// TIA Portal project "TEST_VENDRAME_ALESSANDRO" (V15)

(* hardware
DEVICE "S7-1200 station_1"  S7-1200 Station
   slot 0: "Rack_0"  S7-1200 Rack  Rack  V1.0
   slot 1: "PLC_1"  CPU 1215C DC/DC/DC  6ES7 215-1AG40-0XB0  V4.2
DEVICE "HMI_2"  KTP700 Basic PN
   slot 0: "HMI_2"  KTP700 Basic PN  6AV2 123-2GB03-0AX0  15.0.0.0
   slot 1: "HMI_RT_2"  KTP700 Basic PN  6AV2 123-2GB03-0AX0  15.0.0.0
   slot 5: "HMI_2.IE_CP_1"  PROFINET Interface  15.0.0.0
      slot 1: "PROFINET Interface_1"  PROFINET Interface
         slot 1: "Port_1"  Port
*)

// ===== PLC "PLC_1"  CPU 1215C DC/DC/DC =====

VAR_GLOBAL   // PLC tag table "Default tag table"
   "Clock_Byte" AT %MB666 : Byte;
   "1Hz_Clock" AT %M666.5 : Bool;
   "Clock_5Hz" AT %M666.1 : Bool;
   "Clock_2.5Hz" AT %M666.2 : Bool;
   "Clock_2Hz" AT %M666.3 : Bool;
   "Clock_1.25Hz" AT %M666.4 : Bool;
   "Clock_1Hz" AT %M666.5 : Bool;
   "Clock_0.625Hz" AT %M666.6 : Bool;
   "Clock_0.5Hz" AT %M666.7 : Bool;
END_VAR

DATA_BLOCK "GARA"   // DB1
{ S7_Optimized_Access := 'TRUE' }
VERSION : 0.1
   VAR
      TIMER_START : Bool;
      TIMER_STOP : Bool;
      TIMER_RESET : Bool;
      TIMER_TIME : Real;
      TEMPO_ATLETA_1 : Real;
      TEMPO_ATLETA_2 : Real;
      TEMPO_ATLETA_3 : Real;
      TEMPO_ATLETA_4 : Real;
      TEMPO_ATLETA_5 : Real;
      TEMPO_ATLETA_6 : Real;
      TEMPO_ATLETA_7 : Real;
      TEMPO_ATLETA_8 : Real;
      TimerStop_Atleta_1 : Bool;
      TimerStop_Atleta_2 : Bool;
      TimerStop_Atleta_3 : Bool;
      TimerStop_Atleta_4 : Bool;
      TimerStop_Atleta_5 : Bool;
      TimerStop_Atleta_6 : Bool;
      TimerStop_Atleta_7 : Bool;
      TimerStop_Atleta_8 : Bool;
      Race_Time : Real;
   END_VAR
BEGIN
END_DATA_BLOCK

ORGANIZATION_BLOCK "Main"   // OB1, LAD, ProgramCycle
TITLE = "Main Program Sweep (Cycle)"
{ S7_Optimized_Access := 'TRUE' }
VERSION : 0.1
   VAR_INPUT
      Initial_Call : Bool;   // Initial call of this OB
      Remanence : Bool;   // =True, if remanent data are available
   END_VAR
BEGIN

REGION Network 1
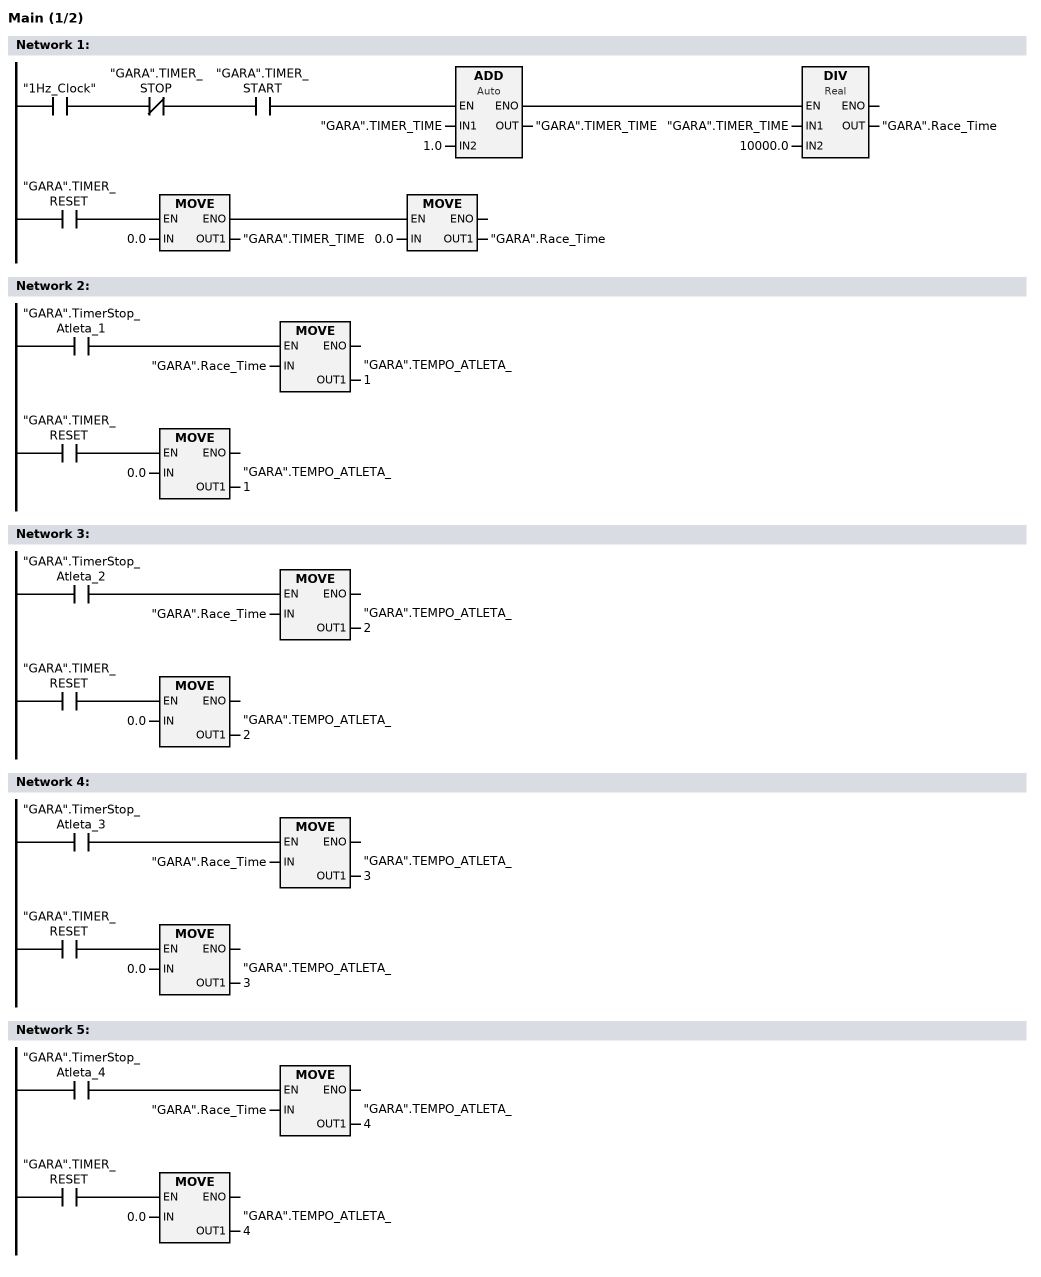
   RUNG wire#powerrail
      Contact( "1Hz_Clock" )
      I_Contact( "GARA".TIMER_STOP )
      Contact( "GARA".TIMER_START )
      Add(in1 := "GARA".TIMER_TIME, in2 := 1.0, out => "GARA".TIMER_TIME)
      { S7_Templates := "SrcType := Real" } Div(in1 := "GARA".TIMER_TIME, in2 := 10000.0, out => "GARA".Race_Time)
   END_RUNG
   RUNG wire#powerrail
      Contact( "GARA".TIMER_RESET )
      Move(in := 0.0, out1 => "GARA".TIMER_TIME)
      Move(in := 0.0, out1 => "GARA".Race_Time)
   END_RUNG
   // the same network as SCL:
   IF "1Hz_Clock" AND NOT "GARA".TIMER_STOP AND "GARA".TIMER_START THEN
       "GARA".TIMER_TIME := "GARA".TIMER_TIME + 1.0;
       "GARA".Race_Time := "GARA".TIMER_TIME / 10000.0;
   END_IF;
   IF "GARA".TIMER_RESET THEN
       "GARA".TIMER_TIME := 0.0;
       "GARA".Race_Time := 0.0;
   END_IF;
END_REGION

REGION Network 2
   RUNG wire#powerrail
      Contact( "GARA".TimerStop_Atleta_1 )
      Move(in := "GARA".Race_Time, out1 => "GARA".TEMPO_ATLETA_1)
   END_RUNG
   RUNG wire#powerrail
      Contact( "GARA".TIMER_RESET )
      Move(in := 0.0, out1 => "GARA".TEMPO_ATLETA_1)
   END_RUNG
   // the same network as SCL:
   IF "GARA".TimerStop_Atleta_1 THEN "GARA".TEMPO_ATLETA_1 := "GARA".Race_Time; END_IF;
   IF "GARA".TIMER_RESET THEN "GARA".TEMPO_ATLETA_1 := 0.0; END_IF;
END_REGION

REGION Network 3
   RUNG wire#powerrail
      Contact( "GARA".TimerStop_Atleta_2 )
      Move(in := "GARA".Race_Time, out1 => "GARA".TEMPO_ATLETA_2)
   END_RUNG
   RUNG wire#powerrail
      Contact( "GARA".TIMER_RESET )
      Move(in := 0.0, out1 => "GARA".TEMPO_ATLETA_2)
   END_RUNG
   // the same network as SCL:
   IF "GARA".TimerStop_Atleta_2 THEN "GARA".TEMPO_ATLETA_2 := "GARA".Race_Time; END_IF;
   IF "GARA".TIMER_RESET THEN "GARA".TEMPO_ATLETA_2 := 0.0; END_IF;
END_REGION

REGION Network 4
   RUNG wire#powerrail
      Contact( "GARA".TimerStop_Atleta_3 )
      Move(in := "GARA".Race_Time, out1 => "GARA".TEMPO_ATLETA_3)
   END_RUNG
   RUNG wire#powerrail
      Contact( "GARA".TIMER_RESET )
      Move(in := 0.0, out1 => "GARA".TEMPO_ATLETA_3)
   END_RUNG
   // the same network as SCL:
   IF "GARA".TimerStop_Atleta_3 THEN "GARA".TEMPO_ATLETA_3 := "GARA".Race_Time; END_IF;
   IF "GARA".TIMER_RESET THEN "GARA".TEMPO_ATLETA_3 := 0.0; END_IF;
END_REGION

REGION Network 5
   RUNG wire#powerrail
      Contact( "GARA".TimerStop_Atleta_4 )
      Move(in := "GARA".Race_Time, out1 => "GARA".TEMPO_ATLETA_4)
   END_RUNG
   RUNG wire#powerrail
      Contact( "GARA".TIMER_RESET )
      Move(in := 0.0, out1 => "GARA".TEMPO_ATLETA_4)
   END_RUNG
   // the same network as SCL:
   IF "GARA".TimerStop_Atleta_4 THEN "GARA".TEMPO_ATLETA_4 := "GARA".Race_Time; END_IF;
   IF "GARA".TIMER_RESET THEN "GARA".TEMPO_ATLETA_4 := 0.0; END_IF;
END_REGION

REGION Network 6
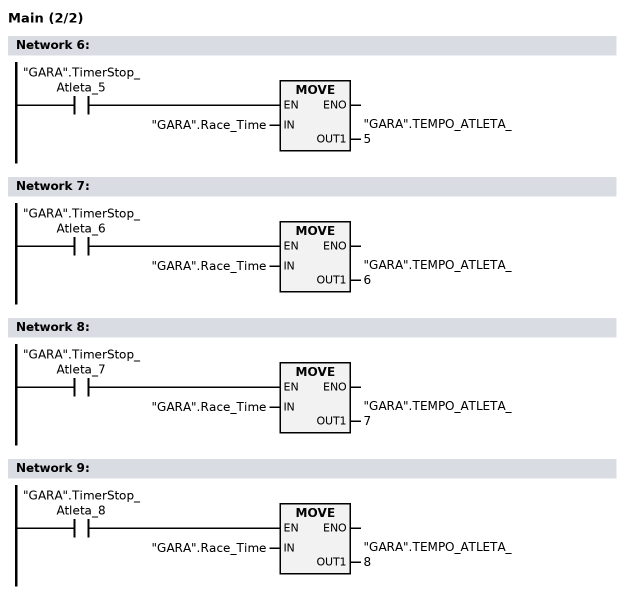
   RUNG wire#powerrail
      Contact( "GARA".TimerStop_Atleta_5 )
      Move(in := "GARA".Race_Time, out1 => "GARA".TEMPO_ATLETA_5)
   END_RUNG
   // the same network as SCL:
   IF "GARA".TimerStop_Atleta_5 THEN "GARA".TEMPO_ATLETA_5 := "GARA".Race_Time; END_IF;
END_REGION

REGION Network 7
   RUNG wire#powerrail
      Contact( "GARA".TimerStop_Atleta_6 )
      Move(in := "GARA".Race_Time, out1 => "GARA".TEMPO_ATLETA_6)
   END_RUNG
   // the same network as SCL:
   IF "GARA".TimerStop_Atleta_6 THEN "GARA".TEMPO_ATLETA_6 := "GARA".Race_Time; END_IF;
END_REGION

REGION Network 8
   RUNG wire#powerrail
      Contact( "GARA".TimerStop_Atleta_7 )
      Move(in := "GARA".Race_Time, out1 => "GARA".TEMPO_ATLETA_7)
   END_RUNG
   // the same network as SCL:
   IF "GARA".TimerStop_Atleta_7 THEN "GARA".TEMPO_ATLETA_7 := "GARA".Race_Time; END_IF;
END_REGION

REGION Network 9
   RUNG wire#powerrail
      Contact( "GARA".TimerStop_Atleta_8 )
      Move(in := "GARA".Race_Time, out1 => "GARA".TEMPO_ATLETA_8)
   END_RUNG
   // the same network as SCL:
   IF "GARA".TimerStop_Atleta_8 THEN "GARA".TEMPO_ATLETA_8 := "GARA".Race_Time; END_IF;
END_REGION
END_ORGANIZATION_BLOCK

(* ===== HMI "HMI_RT_2" =====
system functions are stored by id; their names below are inferred from use
connection "HMI_Connection_1": ETHERNET, SMART_S7_1200_OMS

HMI tags "Default tag table"
   "GARA_TIMER_START" : Bool = PLC GARA.TIMER_START, 1 s
   "GARA_TIMER_RESET" : Bool = PLC GARA.TIMER_RESET, 1 s
   "GARA_TIMER_TIME" : Real = PLC GARA.TIMER_TIME, 1 s
   "GARA_Race_Time" : Real = PLC GARA.Race_Time, 1 s
   "GARA_TIMER_STOP" : Bool = PLC GARA.TIMER_STOP, 1 s
   "GARA_TimerStop_Atleta_1" : Bool = PLC GARA.TimerStop_Atleta_1, 1 s
   "GARA_TEMPO_ATLETA_1" : Real = PLC GARA.TEMPO_ATLETA_1, 1 s
   "GARA_TEMPO_ATLETA_2" : Real = PLC GARA.TEMPO_ATLETA_2, 1 s
   "GARA_TEMPO_ATLETA_3" : Real = PLC GARA.TEMPO_ATLETA_3, 1 s
   "GARA_TEMPO_ATLETA_4" : Real = PLC GARA.TEMPO_ATLETA_4, 1 s
   "GARA_TimerStop_Atleta_2" : Bool = PLC GARA.TimerStop_Atleta_2, 1 s
   "GARA_TimerStop_Atleta_3" : Bool = PLC GARA.TimerStop_Atleta_3, 1 s
   "GARA_TimerStop_Atleta_4" : Bool = PLC GARA.TimerStop_Atleta_4, 1 s

screen "Screen0" 800x480, template "Template_1"
   TextField "HmiScreenItemData" at 80,200 size 640x25; Text 'Screen0'
   Button "Back" at 1,1 size 159x47; TextOff 'Back'
      on Release: ActivateScreen("Root screen", 0)

screen "Root screen" 800x480, template "Template_1"
   TextField "Text field_1" at 9,105 size 67x18; Text 'ATLETA 1:'
   TextField "Text field_2" at 9,135 size 67x18; Text 'ATLETA 2:'
   TextField "Text field_3" at 9,164 size 67x18; Text 'ATLETA 3:'
   IOField "I/O field_1" at 82,104 size 96x23; FormatPattern 99.9
      ProcessValue <- "GARA_TEMPO_ATLETA_1"
   IOField "I/O field_2" at 82,134 size 96x23; FormatPattern 99.9
      ProcessValue <- "GARA_TEMPO_ATLETA_2"
   IOField "I/O field_3" at 82,163 size 96x23; FormatPattern 99.9
      ProcessValue <- "GARA_TEMPO_ATLETA_3"
   TextField "Text field_4" at 10,192 size 67x18; Text 'ATLETA 4:'
   IOField "I/O field_4" at 83,192 size 96x23; FormatPattern 99.9
      ProcessValue <- "GARA_TEMPO_ATLETA_4"
   TextField "Text field_5" at 15,56 size 49x18; Text 'TEMPO:'
   IOField "I/O field_5" at 82,55 size 96x23; FormatPattern 99.99
      ProcessValue <- "GARA_Race_Time"
   Button "Button_1" at 180,51 size 96x32; TextOff 'START'
      on Press: SetBit("GARA_TIMER_START"); ResetBit("GARA_TIMER_RESET"); ResetBit("GARA_TIMER_STOP")
   Button "Button_2" at 372,51 size 96x32; TextOff 'RESET'
      on Press: SetBit("GARA_TIMER_RESET"); ResetBit("GARA_TIMER_START"); ResetBit("GARA_TIMER_STOP")
   TextField "HmiScreenItemData" at 75,2 size 512x22; Text 'GARA 100 m'
   Button "Button_3" at 276,51 size 96x32; TextOff 'STOP'
      on Press: SetBit("GARA_TIMER_STOP"); ResetBit("GARA_TIMER_START"); ResetBit("GARA_TIMER_RESET")
   Button "Button_4" at 180,104 size 96x21; TextOff 'ARRIVATO'
      on Press: function_b14e0dd5("GARA_TimerStop_Atleta_1", 0)
   Button "Button_5" at 180,135 size 96x21; TextOff 'ARRIVATO'
      on Press: function_b14e0dd5("GARA_TimerStop_Atleta_2", 0)
   Button "Button_6" at 180,164 size 96x21; TextOff 'ARRIVATO'
      on Press: function_b14e0dd5("GARA_TimerStop_Atleta_3", 0)
   Button "Button_7" at 180,192 size 96x21; TextOff 'ARRIVATO'
      on Press: function_b14e0dd5("GARA_TimerStop_Atleta_4", 0)

Template "Template_1" 800x480
   Button "Exit" at 714,429 size 71x50; TextOff 'Exit'; PictureOff "ExitRuntime_KTP700_Basic_PN_TR"; PictureOn "ExitRuntime_KTP700_Basic_PN_TR"
      on Release: StopRuntime(0)
   Button "Template_Button" at 614,429 size 71x50; TextOff 'Text'
   Button "Template_Button_1" at 514,429 size 71x50; TextOff 'Text'
   Button "Template_Button_2" at 414,429 size 71x50; TextOff 'Text'
   Button "Template_Button_3" at 314,429 size 71x50; TextOff 'Text'
   Button "Template_Button_4" at 214,429 size 71x50; TextOff 'Text'
   Button "Template_Button_5" at 114,429 size 71x50; TextOff 'Text'
   Button "Start screen" at 14,429 size 71x50; TextOff 'Start screen'; PictureOff "NavigateHome_KTP700_Basic_PN_TR"; PictureOn "NavigateHome_KTP700_Basic_PN_TR"
      on Release: ActivateScreen("Root screen", 0)
*)